// TIA Portal V17 export
// export: Created 2021-12-03T08:13:09.7344415Z, ExportSetting WithDefaults, DisplayName Totally Integrated Automation Portal, DisplayVersion V17, DisplayName TIA Portal Openness, DisplayVersion V17, DisplayName TIA Portal Version Control Interface, DisplayVersion V17, DisplayName STEP 7 Professional, DisplayVersion V17, DisplayName STEP 7 Safety, DisplayVersion V17, DisplayName WinCC Advanced, DisplayVersion V17
FUNCTION_BLOCK "Main_Safety_RTG1"   // FB2, F_FBD
VERSION : 0.1
// stored: AutoNumber false, IsIECCheckEnabled false, UDAEnableTagReadback false
BEGIN

REGION Network 2: Вспомогательные флаги
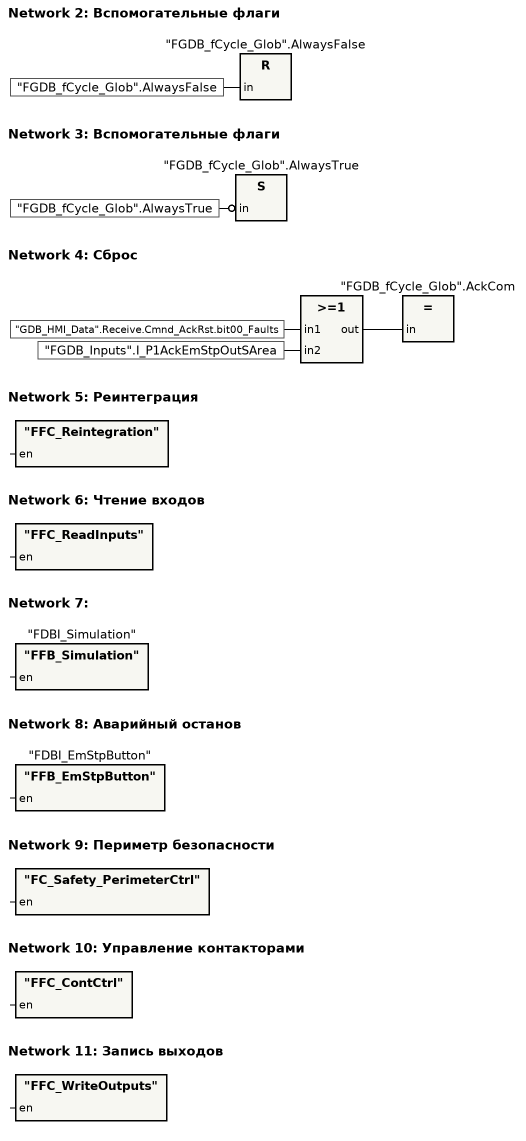
   IF "FGDB_fCycle_Glob".AlwaysFalse THEN "FGDB_fCycle_Glob".AlwaysFalse := FALSE; END_IF;
END_REGION

REGION Network 3: Вспомогательные флаги
   IF NOT "FGDB_fCycle_Glob".AlwaysTrue THEN "FGDB_fCycle_Glob".AlwaysTrue := TRUE; END_IF;
END_REGION

REGION Network 4: Сброс
   "FGDB_fCycle_Glob".AckCom := "GDB_HMI_Data".Receive.Cmnd_AckRst.bit00_Faults OR "FGDB_Inputs".I_P1AckEmStpOutSArea;
END_REGION

REGION Network 5: Реинтеграция
   "FFC_Reintegration"();
END_REGION

REGION Network 6: Чтение входов
   "FFC_ReadInputs"();
END_REGION

REGION Network 7
   "FDBI_Simulation"();   // "FFB_Simulation"
END_REGION

REGION Network 8: Аварийный останов
   "FDBI_EmStpButton"();   // "FFB_EmStpButton"
END_REGION

REGION Network 9: Периметр безопасности
   "FC_Safety_PerimeterCtrl"();
END_REGION

REGION Network 10: Управление контакторами
   "FFC_ContCtrl"();
END_REGION

REGION Network 11: Запись выходов
   "FFC_WriteOutputs"();
END_REGION
END_FUNCTION_BLOCK
